{attribute addProperty BoxType "KL9900-0057"}
{attribute addProperty Id "Channel_1Channel_646A3FAD00"}
{attribute addProperty CRC "3969081270"}
{attribute addProperty SizeInBites "0"}
{attribute addProperty SizeInBytes "0"}
TYPE KL_EC935FB6 :
STRUCT
	{attribute addProperty Name "Channel_1"}
	Channel_1 : Channel_646A3FAD;
END_STRUCT
END_TYPE

(* stored: Version 1.2.0.0, ProductVersion 3.1.4024.9
   DUT KL_EC935FB6: Id {ef57f51c-3d80-49f9-a75b-8eeec76f5243} *)
